(* IEC 61131-3 sources: AXOpen/src/messaging/ctrl/src/Logger, 1 file *)

(* ---- AxoLogger.st ---- *)
USING AXOpen.Core;
USING AXOpen.Messaging;

NAMESPACE AXOpen.Messaging
    CLASS PUBLIC LogEntry
        VAR PUBLIC
            Message : STRING[254];
            Level : eLogLevel;
            Sender : ULINT;
            ToDequeue : BOOL;
        END_VAR
    END_CLASS

    CLASS PUBLIC AxoLogger IMPLEMENTS IAxoLogger
        VAR PUBLIC
            LogEntries : ARRAY[0..100] OF LogEntry;
            Carret : INT := 0;
        END_VAR

        METHOD PUBLIC Log
            VAR_INPUT
                _message : STRING[254];
                _level : eLogLevel := eLogLevel#Information;
                _sender : IAxoObject;
            END_VAR

            IF(Carret > 100) THEN
                Carret := 0;
            END_IF;

            LogEntries[Carret].Message := _message;
            LogEntries[Carret].Level := _level;
            IF(_sender <> NULL) THEN
                LogEntries[Carret].Sender := _sender.GetIdentity();
            END_IF;
            LogEntries[Carret].ToDequeue := TRUE;
            Carret := Carret + 1;

        END_METHOD
    END_CLASS
END_NAMESPACE
